(* Comp A TCP Server*)
FUNCTION_BLOCK FB_ServerApplication
VAR_IN_OUT
	fbTx 			: FB_FrameFifo;(* TX fifo *)
	fbRx 			: FB_FrameFifo;(* RX fifo *)
	fbLog			: FB_LogFifo;(* Log message fifo *)
END_VAR
VAR
	stToClient		: ST_ApplicationBinaryData; (* Tx user data *)
	stFromClient	: ST_ApplicationBinaryData; (* Rx user data *)
	stTxFrame		: ST_BinaryFrame;(* Tx frame buffer (inclusive header) *)
	stRxFrame		: ST_BinaryFrame;(* Rx frame buffer (inclusive header) *)
	state: INT := 0;
	CompBData: LREAL;(* 8 byte *)
	nStateTPC: INT := 0;
END_VAR
VAR PERSISTENT
	ToggleCount: INT := 0;
END_VAR
VAR CONSTANT
	nToogleCycle: INT := 5;
END_VAR

REPEAT		
	(*TPC States* - State Machine Implementation*)	
	CASE nStateTPC OF
	0:(* CLOSED STATE *)
	    stFromClient := fbRx.stGet;  (*RECEIVE SYN*)
		IF ( stFromClient.fpos  <> 0) THEN
			stFromClient.fpos :=HEXSTR_TO_DATA('000007D0', ADR( stFromClient.fpos ), SIZEOF( stFromClient.fpos ) ); (* SEND SYN -ACK*)
			fbTx.AddTail( stPut := stToClient );
			stFromClient.fpos := HEXSTR_TO_DATA('000003E9', ADR( stFromClient.fpos ), SIZEOF( stFromClient.fpos ) );
			fbTx.AddTail( stPut := stToClient );			
			state:=1;
		ELSE
			state:=0;
		END_IF
		
	1: (* SYN RECEIVED STATE*)
		stFromClient := fbRx.stGet;
		IF (stFromClient.fpos =  HEXSTR_TO_DATA('000007D1', ADR( stFromClient.fpos ), SIZEOF( stFromClient.fpos ) )) THEN (*RECEIVED ACK *)
			state:=2;
		ELSE
			state:=1;
		END_IF
		
	2: (* ESTABLISHED STATE*)
		 (* Toogle server data every 5*100 ms*)
		 IF(ToggleCount< nToogleCycle) THEN
			stToClient.fpos:=HEXSTR_TO_DATA('88888888', ADR( stFromClient.fpos ), SIZEOF( stFromClient.fpos ) );  
			ToggleCount := ToggleCount +1 ;
		 ELSE
			stToClient.fpos:=HEXSTR_TO_DATA('88888889', ADR( stFromClient.fpos ), SIZEOF( stFromClient.fpos ) );
			ToggleCount := 0;
		 END_IF
		 fbTx.AddTail( stPut := stToClient ); (* send CompA server data*)
		 stFromClient := fbRx.stGet; (* received ACK*)
		 IF ( stFromClient.fpos = HEXSTR_TO_DATA('000007D1', ADR( stFromClient.fpos ), SIZEOF( stFromClient.fpos ) ) ) THEN
			 stFromClient := fbRx.stGet; (* get CompB Client data*)
			 IF ( stFromClient.fpos <> 0 )THEN 
                CompBData :=  stFromClient.fpos;   
				stToClient.fpos :=  HEXSTR_TO_DATA('000007D1', ADR( stFromClient.fpos ), SIZEOF( stFromClient.fpos ) ); (*send ACK*)
				fbTx.AddTail( stPut := stToClient );
			 END_IF
		  END_IF
		  
		  stFromClient := fbRx.stGet; (* received FIN*)	  
		  IF ( stFromClient.fpos=  HEXSTR_TO_DATA('000003E8', ADR( stFromClient.fpos ), SIZEOF( stFromClient.fpos ) ) )THEN    (* send ACK for client data *)
				stToClient.fpos :=  HEXSTR_TO_DATA('000003E9', ADR( stFromClient.fpos ), SIZEOF( stFromClient.fpos ) );
				fbTx.AddTail( stPut := stToClient );
				state:=3;
		  ELSE
			  state:=2;
		  END_IF
	
	3:  (* CLOSE WAIT STATE*)
		 stToClient.fpos := HEXSTR_TO_DATA('000003E9', ADR( stFromClient.fpos ), SIZEOF( stFromClient.fpos ) );   (* send FIN  for close *)
		 fbTx.AddTail( stPut := stToClient );
		 state :=4;
	
	
	4:  (* LAST ACK STATE*)
		 stFromClient := fbRx.stGet;
		 IF (stFromClient.fpos = HEXSTR_TO_DATA('000005BF', ADR( stFromClient.fpos ), SIZEOF( stFromClient.fpos ) ) ) THEN
			state:=0;	 
		 END_IF
	
	END_CASE
	
UNTIL NOT fbRx.bOk
END_REPEAT

END_FUNCTION_BLOCK

(* stored: Version 1.1.0.1, ProductVersion 3.1.4024.12
   POU FB_ServerApplication: Id {27aa47e1-a593-472a-a33b-33b9fe6bd70e}, SpecialFunc None *)
